Fanuc KAREL source: kt00649.compact.KL

PROGRAM KT00649
%STACKSIZE=65535
%PRIORITY=65535
%NOLOCKGROUP
VAR
H1 : ARRAY[2] OF SHORT
H2 : ARRAY[2] OF SHORT
OUT : INTEGER
BEGIN
H1[1]=2
H2[1]=3
H1[1]=2
H2[1]=3
OUT=(-H1[1])
END KT00649
